PROGRAM PRG_Testing
VAR
	digitalLamp_Wrapper: DigitalLamp_Wrapper;
	digitalLamp_Wrapper2: DigitalLamp_Wrapper;
	
	digitalLampWithPushButton_1: DigitalLampWithPushButton_1;
	digitalLampWithPushButton: OnOffDeviceControl;
	
	analogDevice: AnalogDevice(0, 100, 0, 32767, 10);
	analogStatus: INT;
	setAnalogValue: INT;
	bSetValue: BOOL;
	bInc: BOOL;
	bDec: BOOL;
	bOn: BOOL;
	bOff: BOOL;
	analogDeviceControl: AnalogDeviceControl(ZeroIn:= 0, ZeroOut:= 100, SpanIn:= 0, SpanOut:= 32767, PLC_CYCLE_TIME_ms:= 10, T_LONG_PRESS:= T#2S, RampUpTime:= T#5S, RampDownTime:= T#5S); 
	fan : FourStateDevice;

	fanState: INT := -1;
	fanSpeed: INT;
	
	Variable_In: REAL;			//	raw value of analog card
	Input_min: REAL;			//	min limit of analog card	
	Input_max: REAL;			//	max limit of analog card
	Output_min: REAL;			//	Scalled min limit
	Output_max: REAL;			//	Scalled max limit	
	scalled: REAL;
	
	curtain: Curtain;
	curtainOpening: INT;
	curtainWithSensor: CurtainWithSensor;
	genericCurtain : I_Curtain := CurtainWithSensor;		//	curtain;
	
	bSelectCurtain: BOOL;
	bSelectCurtain2: BOOL;
	simu_tonOpenSensor: TON;
	simu_tonCloseSensor: TON;
	OpenSensor: BOOL;
	CloseSensor: BOOL;
	
	curtainWithManualCalibration: CurtainWithManualCalibration(FALSE);
	simu_Sensor: TIME := T#5s;
END_VAR


	CurtainWithManualCalibration();
	CurtainWithManualCalibration.ClosingTime		:=	simu_Sensor;
	CurtainWithManualCalibration.OpeningTime	:=	simu_Sensor;
	curtainOpening	:=	CurtainWithManualCalibration.Status;
	IF bOn THEN
		CurtainWithManualCalibration.Open(IN := TRUE);
	ELSE
		CurtainWithManualCalibration.Open(IN := FALSE);
	END_IF
	
	IF bOff THEN
		CurtainWithManualCalibration.Close(IN := TRUE);
	ELSE
		CurtainWithManualCalibration.Close(IN := FALSE);
	END_IF	

	
	//CurtainWithSensor(OpenSensor := OpenSensor, CloseSensor := CloseSensor);
//	IF bSelectCurtain THEN
//		genericCurtain	:=	curtain;
//		bSelectCurtain	:=	FALSE;
//	END_IF
//	IF bSelectCurtain2 THEN
//		genericCurtain	:=	curtainWithSensor;
//		bSelectCurtain2	:=	FALSE;
//	END_IF
	
//	curtainOpening	:=	CurtainWithSensor.Status;
//	IF bOn THEN
////		curtain.Open(IN	:=	TRUE);
////		curtainWithSensor.Open(IN	:=	TRUE);
//		genericCurtain.Open(IN	:=	TRUE);
//		simu_tonOpenSensor(IN:= TRUE, PT:= simu_Sensor, Q=> , ET=> );
//		CloseSensor	:= FALSE;
//		IF simu_tonOpenSensor.Q THEN
//			bOn	:=	FALSE;
//			simu_tonOpenSensor(IN:= FALSE);
//			OpenSensor	:=	TRUE;
//		END_IF
//	ELSE
////		curtain.Open(IN	:=	FALSE);
////		curtainWithSensor.Open(IN	:=	FALSE);
//		genericCurtain.Open(IN	:=	FALSE);
//		simu_tonOpenSensor(IN:= FALSE);
//	END_IF
	
//	IF bOff THEN
////		curtain.Close(IN	:=	TRUE);
////		curtainWithSensor.Close(IN	:=	TRUE);
//		genericCurtain.Close(IN	:=	TRUE);
//		simu_tonCloseSensor(IN:= TRUE, PT:= simu_Sensor, Q=> , ET=> );
//		OpenSensor	:=	FALSE;
//		IF simu_tonCloseSensor.Q THEN
//			bOff	:=	FALSE;
//			simu_tonCloseSensor(IN:= FALSE);
//			CloseSensor	:=	TRUE;
//		END_IF
//	ELSE
////		curtain.Close(IN	:=	FALSE);
////		curtainWithSensor.Close(IN	:=	FALSE);
//		genericCurtain.Close(IN	:=	FALSE);
//		simu_tonCloseSensor(IN:= FALSE);
//	END_IF
	


	
//	digitalLamp_Wrapper.KeyType		:=	0;
//	digitalLamp_Wrapper2.KeyType	:=	1;

//	digitalLamp_Wrapper();
//	digitalLamp_Wrapper2();
	
//	digitalLampWithPushButton_1();

//	digitalLampWithPushButton();
	

//	analogDevice();
//	analogStatus	:=	analogDevice.Status;
//	IF bSetValue THEN
//		analogDevice.SetValue(value	:=	setAnalogValue);
//		bSetValue	:=	FALSE;
//	END_IF
	
//	IF bInc THEN
//		analogDevice.IncreaseValue(EN:= TRUE, RampUpTime	:=	T#5S);
//	ELSE
//		analogDevice.IncreaseValue(EN:= FALSE, RampUpTime	:=	T#5S);
//	END_IF
	
//	IF bDec THEN
//		analogDevice.DecreaseValue(EN:= TRUE, RampDownTime	:=	T#5S);
//	ELSE
//		analogDevice.DecreaseValue(EN:= FALSE, RampDownTime	:=	T#5S);
//	END_IF
	
//	IF bOn THEN
//		analogDevice.On();
//	END_IF
	
//	IF bOff THEN
//		analogDevice.Off();
//	END_IF
	
//	analogDeviceControl();
//	analogStatus	:=	analogDeviceControl.Status;
		
//	fan();
//	fanSpeed	:=	fan.Status;
//	IF bOff THEN
//	fan.Off();
//	bOff:=FALSE;
//	END_IF
		
//	IF bOn THEN
//		fan.On();
//		bOn:=FALSE;
//	END_IF
	
//	CASE fanState OF
//	0:	;
//	1:	fan.State_1();
//	2:	fan.State_2();
//	3:	fan.State_3();
//	4:	fan.State_4();
//	END_CASE
	
		
//IF (Input_max - Input_min) <> 0 THEN
//	scalled := ((Variable_In - Input_min) / (Input_max - Input_min)) * (Output_max - Output_min) + Output_min;
//ELSE
//	scalled	:=	0;
//END_IF

END_PROGRAM

(* stored: Version 1.1.0.1, ProductVersion 3.1.4024.13
   POU PRG_Testing: Id {b6fffdb7-2a36-4774-ac1d-63cbacf3b383}, SpecialFunc None *)
